{attribute 'qualified_only'}
VAR_GLOBAL
	
END_VAR

(* stored: Version 1.1.0.1
   GVL GVL_IO: Id {31a5c8d3-3071-4b8b-bc39-ff6bf40b714f} *)
